# EPICS autosave request: support/areaDetector-s55/iocBoot/iocProsilica/auto_settings.req
file "ADBase_settings.req",         P=$(P),  R=cam1:
file "NDFile_settings.req",         P=$(P),  R=cam1:
file "prosilica_settings.req",      P=$(P),  R=cam1:
#file "ADBase_settings.req",         P=$(P),  R=cam2:
#file "NDFile_settings.req",         P=$(P),  R=cam2:
#file "prosilica_settings.req",      P=$(P),  R=cam2:
file "NDPluginBase_settings.req",   P=$(P),  R=image1:
file "NDStdArrays_settings.req",    P=$(P),  R=image1:
file "commonPlugin_settings.req",   P=$(P)
